% RSLogix 500 project Digital-Filling-Station.RSS, saved by version 8.30.00.16 %
PROJECT "UNTITLED"    % processor: Bul.1763 MicroLogix 1100 Series B %

PROGRAM FILES
  LAD 2 "MAIN"  3 rungs
  LAD 3 "IO"  8 rungs  % INPUT/OUTPUT %
  LAD 4 "CTRL"  6 rungs  % CONTROL LOGIC %

DATA FILES
  O0 OUTPUT  4 elements
  I1 INPUT  6 elements
  S2 STATUS  66 elements
  B3 BINARY  4 elements
  T4 TIMER  1 elements
  C5 COUNTER  1 elements
  R6 CONTROL  1 elements
  N7 INTEGER  1 elements
  F8 FLOAT  1 elements

LADDER 2 "MAIN"
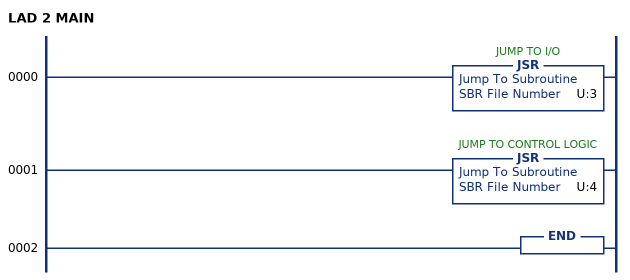
% Rung: 0 %
SOR JSR U:3 EOR
%   U:3  "JUMP TO I/O" %
% Rung: 1 %
SOR JSR U:4 EOR
%   U:4  "JUMP TO CONTROL LOGIC" %
% Rung: 2 %
SOR END EOR

LADDER 3 "IO"    % INPUT/OUTPUT %
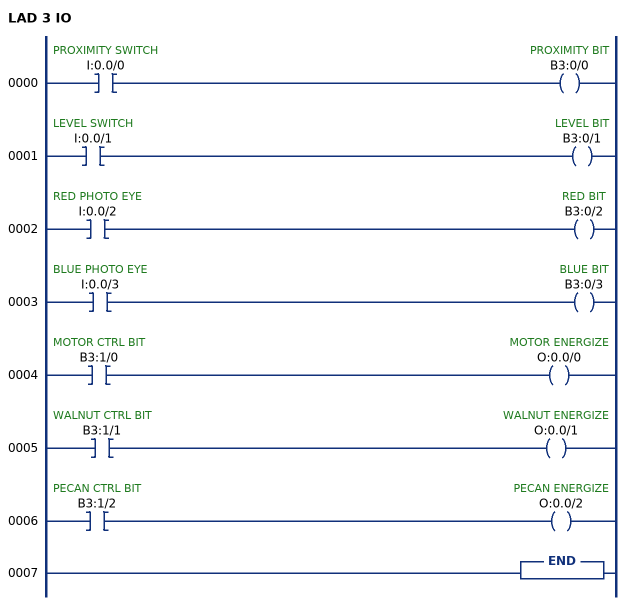
% Rung: 0 %
SOR XIC I:0.0/0 OTE B3:0/0 EOR
%   I:0.0/0  "PROXIMITY SWITCH" %
%   B3:0/0  "PROXIMITY BIT" %
% Rung: 1 %
SOR XIC I:0.0/1 OTE B3:0/1 EOR
%   I:0.0/1  "LEVEL SWITCH" %
%   B3:0/1  "LEVEL BIT" %
% Rung: 2 %
SOR XIC I:0.0/2 OTE B3:0/2 EOR
%   I:0.0/2  "RED PHOTO EYE" %
%   B3:0/2  "RED BIT" %
% Rung: 3 %
SOR XIC I:0.0/3 OTE B3:0/3 EOR
%   I:0.0/3  "BLUE PHOTO EYE" %
%   B3:0/3  "BLUE BIT" %
% Rung: 4 %
SOR XIC B3:1/0 OTE O:0.0/0 EOR
%   B3:1/0  "MOTOR CTRL BIT" %
%   O:0.0/0  "MOTOR ENERGIZE" %
% Rung: 5 %
SOR XIC B3:1/1 OTE O:0.0/1 EOR
%   B3:1/1  "WALNUT CTRL BIT" %
%   O:0.0/1  "WALNUT ENERGIZE" %
% Rung: 6 %
SOR XIC B3:1/2 OTE O:0.0/2 EOR
%   B3:1/2  "PECAN CTRL BIT" %
%   O:0.0/2  "PECAN ENERGIZE" %
% Rung: 7 %
SOR END EOR

LADDER 4 "CTRL"    % CONTROL LOGIC %
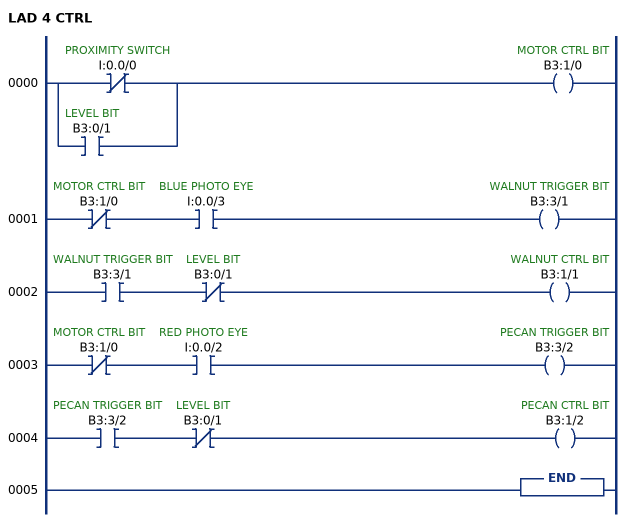
% Rung: 0 %
SOR BST XIO I:0.0/0 NXB XIC B3:0/1 BND OTE B3:1/0 EOR
%   I:0.0/0  "PROXIMITY SWITCH" %
%   B3:0/1  "LEVEL BIT" %
%   B3:1/0  "MOTOR CTRL BIT" %
% Rung: 1 %
SOR XIO B3:1/0 XIC I:0.0/3 OTE B3:3/1 EOR
%   B3:1/0  "MOTOR CTRL BIT" %
%   I:0.0/3  "BLUE PHOTO EYE" %
%   B3:3/1  "WALNUT TRIGGER BIT" %
% Rung: 2 %
SOR XIC B3:3/1 XIO B3:0/1 OTE B3:1/1 EOR
%   B3:3/1  "WALNUT TRIGGER BIT" %
%   B3:0/1  "LEVEL BIT" %
%   B3:1/1  "WALNUT CTRL BIT" %
% Rung: 3 %
SOR XIO B3:1/0 XIC I:0.0/2 OTE B3:3/2 EOR
%   B3:1/0  "MOTOR CTRL BIT" %
%   I:0.0/2  "RED PHOTO EYE" %
%   B3:3/2  "PECAN TRIGGER BIT" %
% Rung: 4 %
SOR XIC B3:3/2 XIO B3:0/1 OTE B3:1/2 EOR
%   B3:3/2  "PECAN TRIGGER BIT" %
%   B3:0/1  "LEVEL BIT" %
%   B3:1/2  "PECAN CTRL BIT" %
% Rung: 5 %
SOR END EOR

OTHER DOCUMENTED ADDRESSES
  B3:3/0  "MOTOR TRIGGER BIT"
  I:1.0/0  "PROXIMITY BIT"
  I:1.0/1  "LEVEL BIT"
  I:1.0/2  "RED BIT"
  I:1.0/3  "BLUE BIT"
